PROPERTY proOnY_ITF : CtaSysIO.ITF_IO
GET
END_GET
END_PROPERTY

PROPERTY proIsRegulatet : BOOL
GET
END_GET
END_PROPERTY

PROPERTY proIsHandOnOrOff : BOOL
GET
END_GET
END_PROPERTY

PROPERTY proRunAfterTimeAktive : BOOL
GET
END_GET
END_PROPERTY

PROPERTY proLeadTimeAktive : BOOL
GET
END_GET
END_PROPERTY

PROPERTY proIsReady : BOOL
GET
END_GET
END_PROPERTY

PROPERTY proAuto : BOOL
GET
END_GET
SET
END_SET
END_PROPERTY

PROPERTY proHandOn : BOOL
SET
END_SET
GET
END_GET
END_PROPERTY

PROPERTY proIsError : BOOL
GET
END_GET
END_PROPERTY

PROPERTY proIsWarning : BOOL
GET
END_GET
END_PROPERTY

PROPERTY proEn : BOOL
GET
END_GET
SET
END_SET
END_PROPERTY

PROPERTY proHardWareHandModulAktive : BOOL
GET
END_GET
END_PROPERTY

PROPERTY proIsEnabled : BOOL
GET
END_GET
END_PROPERTY

PROPERTY proMotorIsOn : BOOL
GET
END_GET
END_PROPERTY

PROPERTY proHandOff : BOOL
SET
END_SET
GET
END_GET
END_PROPERTY

PROPERTY proRevisionSwitchOk : BOOL
GET
END_GET
END_PROPERTY

PROPERTY proHandOnY : REAL
SET
END_SET
GET
END_GET
END_PROPERTY

{attribute 'hide'} 
PROPERTY INTERNAL proEnSymbol : STRING
GET
END_GET
END_PROPERTY

PROPERTY proIsOn : BOOL
GET
END_GET
END_PROPERTY

PROPERTY proIsOnY : REAL
GET
END_GET
END_PROPERTY

PROPERTY proLeadTime : TIME
GET
END_GET
END_PROPERTY

PROPERTY proOn : BOOL
GET
END_GET
END_PROPERTY

PROPERTY proOnY : REAL
GET
END_GET
END_PROPERTY

PROPERTY proRunAfterTime : TIME
GET
END_GET
END_PROPERTY

{attribute 'hide'} 
PROPERTY INTERNAL proStateSymbol : STRING
GET
END_GET
END_PROPERTY

{attribute 'monitoring' := 'variable'}
PROPERTY proLockDown : BOOL
GET
END_GET
END_PROPERTY

{attribute 'monitoring' := 'variable'}
PROPERTY proAvailable : BOOL
GET
END_GET
END_PROPERTY

{attribute 'monitoring' := 'variable'}
PROPERTY proAcknowlege : BOOL
GET
END_GET
END_PROPERTY

PROPERTY proIconNr : UINT
SET
END_SET
GET
END_GET
END_PROPERTY

END_INTERFACE

// 30 Program Organization Units/fcGetBigerStringValue
FUNCTION fcGetBigerStringValue : INT
VAR_INPUT
    st1     :   STRING(255);
    st2     :   STRING(255);
END_VAR
VAR
    diFor: DINT;
    diMax: DINT;
END_VAR

IF LEN(st1) > LEN(st2) THEN
    diMax := LEN(st2); 
    fcGetBigerStringValue := 1;
ELSIF LEN(st1) < LEN(st2) THEN
    diMax := LEN(st1);
    fcGetBigerStringValue := 2;     
ELSE
    diMax := LEN(st1);    
END_IF;
FOR diFor := 0 TO  diMax DO
    IF st1[diFor] > st2[diFor] THEN
        fcGetBigerStringValue := 1;  
        EXIT; 
    ELSIF st1[diFor] < st2[diFor] THEN
        fcGetBigerStringValue := 2;  
        EXIT;
    END_IF;
END_FOR;

END_FUNCTION

// 30 Program Organization Units/fcCheckQuerryAndIconReturn
FUNCTION fcCheckQuerryAndIconReturn : BOOL
VAR_INPUT
	_ITF_IN			: 	ITF_ANTRIEB;
	_uiIconNr_IN	:	UINT;
END_VAR

IF __QUERYINTERFACE(_ITF_IN,_ITF_IN) THEN
	fcCheckQuerryAndIconReturn := TRUE;	
	_ITF_IN.proIconNr := _uiIconNr_IN;
ELSE
	fcCheckQuerryAndIconReturn :=  FALSE;
END_IF

END_FUNCTION

// 40 Visualizations/POPUP/POPUP_ANTRIEB
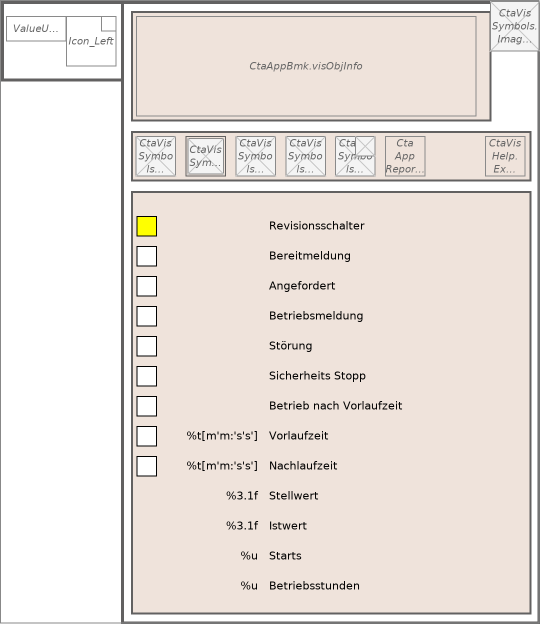
VISUALIZATION POPUP_ANTRIEB  // 540x624
VAR_INPUT
    ITF_ANTRIEBIN    	:   ITF_ANTRIEB;
	stExklParameter_IN	:	STRING[40];	
	uiPopUpGruppe 		: 	UINT;
END_VAR
    RoundedRectangle (1,1 160x80)
    RoundedRectangle (121,1 419x623)
    RoundedRectangle (131,11 360x110)
    Frame (136,16 340x100)
        shows CtaAppBmk.visObjInfo(ITF_BMK_IN := ITF_ANTRIEBIN)
    Image (490,1 50x50), image: CtaVisSymbols.ImagePool.close_solo_black
        OnMouseClick:  Dialog=POPUP_ANTRIEB, Result=None, NumpadKeypadSet=True
    Frame (6,16 110x50), input disabled if: TRUE, frame switch variable: ITF_ANTRIEBIN.proIconNr
        shows VIS_ANTRIEB_LEFT_ABOVE(ITF_ANTRIEB_IN := ITF_ANTRIEBIN, stExklParameter := stExklParameter_IN)
        shows VIS_ANTRIEB_LEFT_BELOW(ITF_ANTRIEB_IN := ITF_ANTRIEBIN, stExklParameter := stExklParameter_IN)
        shows VIS_ANTRIEB_RIGHT_ABOVE(ITF_ANTRIEB_IN := ITF_ANTRIEBIN, stExklParameter := stExklParameter_IN)
        shows VIS_ANTRIEB_RIGHT_BELOW(ITF_ANTRIEB_IN := ITF_ANTRIEBIN, stExklParameter := stExklParameter_IN)
    RoundedRectangle (131,191 400x423)
    Frame (132,206 398x400), frame switch variable: uiPopUpGruppe
        shows VIS_ANTRIEB_OVERVIEW(ITF_ANTRIEBIN := ITF_ANTRIEBIN)
        shows VIS_ANTRIEB_MANUAL(ITF_ANTRIEBIN := ITF_ANTRIEBIN)
        shows VIS_ANTRIEB_PARAMETER(ITF_ANTRIEBIN := ITF_ANTRIEBIN)
        shows VIS_ANTRIEB_IO(ITF_ANTRIEBIN := ITF_ANTRIEBIN)
        shows AT_BUS(ITF_ANTRIEBIN := ITF_ANTRIEBIN)
        shows VIS_ANTRIEB_REPORTS(ITF_ANTRIEBIN := ITF_ANTRIEBIN)
        pReferences[2]: ITF_Parameter=ITF_ANTRIEBIN.proParameter
    RoundedRectangle (131,131 400x50)
    Frame (131,136 399x40)
        shows VIS_ANTRIEB_LISTE(uiPopUpGruppe := uiPopUpGruppe, xHand := ITF_ANTRIEBIN.proIsHandOnOrOff, xHandOff := ITF_ANTRIEBIN.proHandOff, ITF_REPORTMANAGER_IN := ITF_ANTRIEBIN.proITF_REPORTMANAGER, xBusTestAktiv := ITF_ANTRIEBIN.proModbusTest, stExklParameter_IN := stExklParameter_IN)
    InvisibleInput (131,3 360x48)
END_VISUALIZATION

// 40 Visualizations/POPUP/VIS_ANTRIEB_LISTE
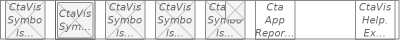
VISUALIZATION VIS_ANTRIEB_LISTE  // 400x40
VAR_IN_OUT
	uiPopUpGruppe 			:	UINT;
END_VAR
VAR_INPUT
    xHand           		: 	BOOL;
    xHandOff        		: 	BOOL;
    ITF_REPORTMANAGER_IN 	: 	CtaAppReport.ITF_REPORTMANAGER;
    xBusTestAktiv   		: 	BOOL;	
	stExklParameter_IN		:	STRING[40];
END_VAR
    Group (5,0 40x40)
        RoundedRectangle (0,0 40x40), colour toggle: uiPopUpGruppe = 0
            OnMouseDown: execute { uiPopUpGruppe := 0; }
        Image (0,0 40x40), image: CtaVisSymbols.ImagePool.eye
            OnMouseDown: execute { uiPopUpGruppe := 0; }
    Group (105,0 40x40)
        RoundedRectangle (0,0 40x40), colour toggle: uiPopUpGruppe = 2
            OnMouseDown: execute { uiPopUpGruppe := 2; }
        Image (0,0 40x40), image: CtaVisSymbols.ImagePool.gear
            OnMouseDown: execute { uiPopUpGruppe := 2; }
    Group (55,0 40x40)
        RoundedRectangle (0,0 40x40), colour toggle: uiPopUpGruppe = 1
            OnMouseDown: execute { uiPopUpGruppe := 1; }
        Image (2,2 36x36), image: CtaVisSymbols.ImagePool.front_hand_Black
            OnMouseDown: execute { uiPopUpGruppe := 1; }
        Image (2,2 36x36), invisible if: NOT xHand, image: CtaVisSymbols.ImagePool.front_hand_Yellow
            OnMouseDown: execute { uiPopUpGruppe := 1; }
        Image (2,2 36x36), invisible if: NOT xHandOff, image: CtaVisSymbols.ImagePool.front_hand_Yellow_Off
            OnMouseDown: execute { uiPopUpGruppe := 1; }
    Group (155,0 40x40)
        RoundedRectangle (0,0 40x40), colour toggle: uiPopUpGruppe = 3
            OnMouseDown: execute { uiPopUpGruppe := 3; }
        Image (0,0 40x40), image: CtaVisSymbols.ImagePool.dip-switch
            OnMouseDown: execute { uiPopUpGruppe := 3; }
    Group (205,0 40x40)
        RoundedRectangle (0,0 40x40), colour toggle: uiPopUpGruppe = 4
            OnMouseDown: execute { uiPopUpGruppe := 4; }
        Image (0,0 40x40), image: CtaVisSymbols.ImagePool.lan
            OnMouseDown: execute { uiPopUpGruppe := 4; }
        Image (20,0 20x20), invisible if: NOT xBusTestAktiv, image: CtaVisSymbols.ImagePool.front_hand_Yellow
            OnMouseDown: execute { uiPopUpGruppe := 4; }
    Group (255,0 40x40)
        RoundedRectangle (0,0 40x40), colour toggle: uiPopUpGruppe = 5
            OnMouseDown: execute { uiPopUpGruppe := 5; }
        Frame (0,0 40x40), input disabled if: TRUE
            shows CtaAppReport.VIS_ANZ_REPORTS_MODUL(ITF_REPORTMANAGER_IN := ITF_REPORTMANAGER_IN)
            OnMouseDown: execute { uiPopUpGruppe := 5; }
    Group (355,0 40x40)
        RoundedRectangle (0,0 40x40), invisible if: stExklParameter_IN = ' '
        Frame (0,0 40x40)
            shows CtaVisHelp.ExkParameterSymbol(stExklParameter := stExklParameter_IN)
END_VISUALIZATION

// 40 Visualizations/ICON/ANTRIEB_RIGHT/ANTRIEB_RIGHT_ABOVE/VIS_ANTRIEB_RigthAboveCheckQuerry
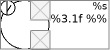
VISUALIZATION VIS_ANTRIEB_RigthAboveCheckQuerry  // 110x50
VAR_INPUT
    ITF_ANTRIEB_IN   :   ITF_ANTRIEB;	
END_VAR
VAR_INPUT
	stExklParameter		:	STRING[40];
END_VAR
    Frame (0,0 110x50)
        shows VIS_ANTRIEB_RigthAboveCheckIsEnabled(ITF_ANTRIEB_IN := ITF_ANTRIEB_IN, stExklParameter := stExklParameter)
END_VISUALIZATION

// 40 Visualizations/ICON/ANTRIEB_RIGHT/ANTRIEB_RIGHT_ABOVE/VIS_ANTRIEB_RIGHT_ABOVE
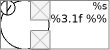
VISUALIZATION VIS_ANTRIEB_RIGHT_ABOVE  // 110x50
VAR_INPUT
    ITF_ANTRIEB_IN   :   ITF_ANTRIEB;	
END_VAR
VAR_INPUT CONSTANT
	stExklParameter		:	STRING[40] := ' ';
END_VAR
VAR CONSTANT
	uiIconNr		: UINT := 2;
END_VAR
    Frame (0,0 110x50), invisible if: NOT fcCheckQuerryAndIconReturn(_ITF_IN := ITF_ANTRIEB_IN, _uiIconNr_IN := uiIconNr)
        shows VIS_ANTRIEB_RigthAboveCheckQuerry(ITF_ANTRIEB_IN := ITF_ANTRIEB_IN, stExklParameter := stExklParameter)
END_VISUALIZATION

// 40 Visualizations/ICON/ANTRIEB_RIGHT/ANTRIEB_RIGHT_ABOVE/VIS_ANTRIEB_RigthAboveCheckIsEnabled
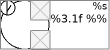
VISUALIZATION VIS_ANTRIEB_RigthAboveCheckIsEnabled  // 110x50
VAR_INPUT
    ITF_ANTRIEB_IN   :   ITF_ANTRIEB;	
END_VAR
VAR_INPUT
	stExklParameter		:	STRING[40];
END_VAR
    Frame (0,0 50x50), invisible if: NOT ITF_ANTRIEB_IN.proIsEnabled
        shows Icon_Right(ITF_ANTRIEB_IN := ITF_ANTRIEB_IN)
        shows Value_Right()
    Frame (50,0 60x25), invisible if: NOT ITF_ANTRIEB_IN.proIsEnabled
        shows ValueUpDwn(ITF_ANTRIEB_IN := ITF_ANTRIEB_IN, uiTextAusrichtung := 4)
    Frame (0,0 15x15), invisible if: NOT ITF_ANTRIEB_IN.proIsEnabled
        shows CommandOn(ITF_ANTRIEB_IN := ITF_ANTRIEB_IN)
    Rectangle (0,0 110x50)
        OnMouseClick:  Dialog=POPUP_ANTRIEB, Parameters={uiPopUpGruppe: 0, stExklParameter_IN: stExklParameter, ITF_ANTRIEBIN: ITF_ANTRIEB_IN}, OpenCentered=True
END_VISUALIZATION

// 40 Visualizations/ICON/ANTRIEB_BASE/CommandOn
VISUALIZATION CommandOn  // 15x15
VAR_INPUT
    ITF_ANTRIEB_IN   :   ITF_ANTRIEB;	
END_VAR
    Ellipse (0,0 15x15), colour toggle: ITF_ANTRIEB_IN.proOn
    Line (7,15) (7,10)
    Line (7,5) (7,0)
    Line (7,11) (11,5), invisible if: ITF_ANTRIEB_IN.proOn
    Line (7,15) (7,0), invisible if: NOT ITF_ANTRIEB_IN.proOn
END_VISUALIZATION

// 40 Visualizations/ICON/ANTRIEB_BASE/ICON/Icon_Left
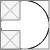
VISUALIZATION Icon_Left  // 50x50
VAR_INPUT
    ITF_ANTRIEB_IN   :   ITF_ANTRIEB;	
END_VAR
    Ellipse (0,0 49x49), colour toggle: ITF_ANTRIEB_IN.proMotorIsOn, invisible if: ITF_ANTRIEB_IN.proIsError
    Ellipse (0,0 49x49), colour toggle: ITF_ANTRIEB_IN.proIsError
    Image (0,0 20x20), invisible if: NOT ITF_ANTRIEB_IN.proIsWarning, image: CtaVisSymbols.ImagePool.CtaWarning
    Image (0,30 20x20), invisible if: NOT ITF_ANTRIEB_IN.proIsHandOnOrOff, image: CtaVisSymbols.ImagePool.front_hand_Yellow
    Image (0,30 20x20), invisible if: NOT ITF_ANTRIEB_IN.proHandOff, image: CtaVisSymbols.ImagePool.front_hand_Yellow_Off
END_VISUALIZATION

// 40 Visualizations/POPUP/PARAMETER/VIS_ANTRIEB_PARAMETER
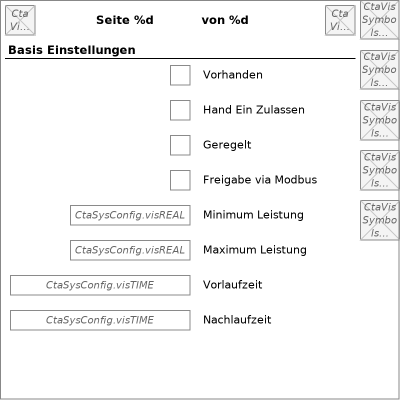
VISUALIZATION VIS_ANTRIEB_PARAMETER  // 400x400
VAR_INPUT
    ITF_ANTRIEBIN    :   ITF_ANTRIEB;	
END_VAR
VAR
    uiParameterGruppe : UINT;
END_VAR
    Frame (360,0 40x300)
        shows VIS_ANTRIEB_PARAMETER_LISTE(uiParameterGruppe := uiParameterGruppe)
    Frame (0,0 360x400), frame switch variable: uiParameterGruppe
        shows VIS_ANTRIEB_PARAMETER_BASE(ITF_ANTRIEBIN := ITF_ANTRIEBIN)
        shows VIS_ANTRIEB_PARAMETER_FUSES(ITF_ANTRIEBIN := ITF_ANTRIEBIN)
        shows VIS_ANTRIEB_PARAMETER_IO(ITF_ANTRIEBIN := ITF_ANTRIEBIN)
        shows VIS_ANTRIEB_PARAMETER_DATA(ITF_ANTRIEBIN := ITF_ANTRIEBIN)
        shows VIS_ANTRIEB_PARAMETER_TRENDLOG(ITF_ANTRIEBIN := ITF_ANTRIEBIN)
        pReferences[0]: ITF_Parameter=ITF_Parameter
        pReferences[1]: ITF_Parameter=ITF_Parameter
        pReferences[2]: ITF_Parameter=ITF_Parameter
        pReferences[3]: ITF_Parameter=ITF_Parameter
        pReferences[4]: ITF_Parameter=ITF_Parameter
END_VISUALIZATION

// 40 Visualizations/POPUP/PARAMETER/VIS_ANTRIEB_PARAMETER_LISTE
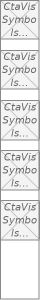
VISUALIZATION VIS_ANTRIEB_PARAMETER_LISTE  // 40x300
VAR_IN_OUT
	uiParameterGruppe : UINT;
END_VAR
    RoundedRectangle (0,150 39x39), colour toggle: uiParameterGruppe = 3
        OnMouseDown: execute { uiParameterGruppe := 3; }
    RoundedRectangle (0,100 39x39), colour toggle: uiParameterGruppe = 2
        OnMouseDown: execute { uiParameterGruppe := 2; }
    RoundedRectangle (0,50 39x39), colour toggle: uiParameterGruppe = 1
        OnMouseDown: execute { uiParameterGruppe := 1; }
    RoundedRectangle (0,0 39x39), colour toggle: uiParameterGruppe = 0
        OnMouseDown: execute { uiParameterGruppe := 0; }
    RoundedRectangle (0,200 39x39), colour toggle: uiParameterGruppe = 4
        OnMouseDown: execute { uiParameterGruppe := 4; }
    Image (0,0 39x39), image: CtaVisSymbols.ImagePool.engine
        OnMouseDown: execute { uiParameterGruppe := 0; }
    Image (0,50 39x39), image: CtaVisSymbols.ImagePool.electric_bolt_24dp_000000_FILL0_wght400_GRAD0_opsz24
        OnMouseDown: execute { uiParameterGruppe := 1; }
    Image (0,100 40x40), image: CtaVisSymbols.ImagePool.dip-switch
        OnMouseDown: execute { uiParameterGruppe := 2; }
    Image (0,150 40x40), image: CtaVisSymbols.ImagePool.database_black
        OnMouseDown: execute { uiParameterGruppe := 3; }
    Image (0,200 40x40), image: CtaVisSymbols.ImagePool.sine-wave
        OnMouseDown: execute { uiParameterGruppe := 4; }
END_VISUALIZATION

// 40 Visualizations/POPUP/MANUAL/VIS_ANTRIEB_MANUAL
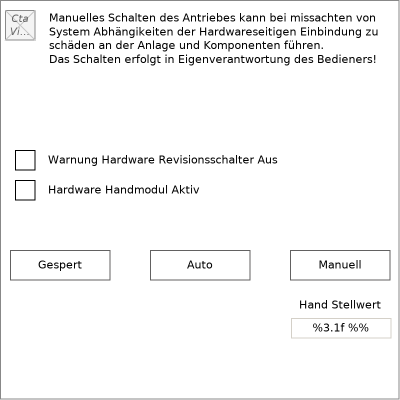
VISUALIZATION VIS_ANTRIEB_MANUAL  // 400x400
VAR_INPUT
    ITF_ANTRIEBIN    :   ITF_ANTRIEB;	
END_VAR
    Label (46,10 350x100), "Manuelles Schalten des Antriebes kann bei missachten von System Abhängikeiten der Hardwareseitigen Einbindung zu schäden an der Anlage und Komponenten führen. Das Schalten erfolgt in Eigenverantwortung des Bedieners!"
    Textfield (291,318 100x20), "%3.1f %%", text variable: ITF_ANTRIEBIN.proHandOnY, invisible if: NOT ITF_ANTRIEBIN.proIsRegulatet
        OnMouseClick: write the text variable via InputWithLimits, min 0, max 100, title 'Stellwert'
    Image (5,10 30x30), image: CtaVisSymbols.ImagePool.CtaWarning
    Label (290,295 100x20), "Hand Stellwert"
    Rectangle (15,180 20x20), colour toggle: ITF_ANTRIEBIN.proHardWareHandModulAktive, invisible if: NOT ITF_ANTRIEBIN.proHardWareHandModulAktive
    Label (45,180 200x20), "Hardware Handmodul Aktiv", invisible if: NOT ITF_ANTRIEBIN.proHardWareHandModulAktive
    Label (45,150 350x20), "Warnung Hardware Revisionsschalter Aus", invisible if: ITF_ANTRIEBIN.proRevisionSwitchOk
    Rectangle (15,150 20x20), colour toggle: NOT ITF_ANTRIEBIN.proRevisionSwitchOk, invisible if: ITF_ANTRIEBIN.proRevisionSwitchOk
    RoundedRectangle (10,250 100x30), "Gespert", colour toggle: ITF_ANTRIEBIN.proHandOff
        toggle ITF_ANTRIEBIN.proHandOff
    RoundedRectangle (150,250 100x30), "Auto", colour toggle: ITF_ANTRIEBIN.proAuto
        toggle ITF_ANTRIEBIN.proAuto
    RoundedRectangle (290,250 100x30), "Manuell", colour toggle: ITF_ANTRIEBIN.proHandOn
        toggle ITF_ANTRIEBIN.proHandOn
END_VISUALIZATION

// 40 Visualizations/POPUP/OVERVIEW/VIS_ANTRIEB_OVERVIEW
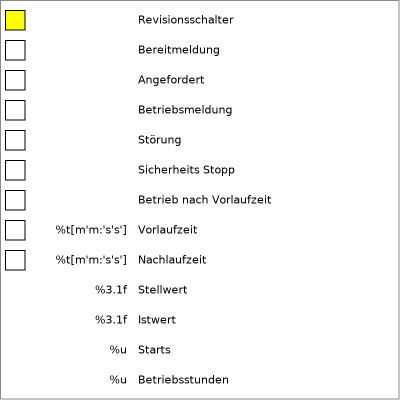
VISUALIZATION VIS_ANTRIEB_OVERVIEW  // 400x400
VAR_INPUT
    ITF_ANTRIEBIN    :   ITF_ANTRIEB;	
END_VAR
    Label (135,220 200x20), "Vorlaufzeit"
    Label (135,250 200x20), "Nachlaufzeit"
    Textfield (30,220 100x20), "%t[m'm:'s's']", text variable: ITF_ANTRIEBIN.proLeadTime
    Textfield (30,250 100x20), "%t[m'm:'s's']", text variable: ITF_ANTRIEBIN.proRunAfterTime
    Rectangle (5,220 20x20), colour toggle: ITF_ANTRIEBIN.proLeadTimeAktive
    Rectangle (5,250 20x20), colour toggle: ITF_ANTRIEBIN.proRunAfterTimeAktive
    Label (135,10 200x20), "Revisionsschalter"
    Label (135,40 200x20), "Bereitmeldung"
    Label (135,100 200x20), "Betriebsmeldung"
    Label (135,130 200x20), "Störung"
    Label (135,70 200x20), "Angefordert"
    Rectangle (5,10 20x20), colour toggle: ITF_ANTRIEBIN.proRevisionSwitchOk
    Rectangle (5,40 20x20), colour toggle: ITF_ANTRIEBIN.proIsReady
    Rectangle (5,70 20x20), colour toggle: ITF_ANTRIEBIN.proOn
    Rectangle (5,100 20x20), colour toggle: ITF_ANTRIEBIN.proMotorIsOn
    Rectangle (5,130 20x20), colour toggle: ITF_ANTRIEBIN.proIsError
    Label (135,160 200x20), "Sicherheits Stopp"
    Rectangle (5,160 20x20)
    Label (135,190 200x20), "Betrieb nach Vorlaufzeit"
    Rectangle (5,190 20x20), colour toggle: ITF_ANTRIEBIN.proIsOn
    Label (135,280 200x20), "Stellwert", invisible if: NOT ITF_ANTRIEBIN.proIsRegulatet
    Label (135,310 200x20), "Istwert", invisible if: NOT ITF_ANTRIEBIN.proIsRegulatet
    Textfield (30,280 100x20), "%3.1f", text variable: ITF_ANTRIEBIN.proOnY, invisible if: NOT ITF_ANTRIEBIN.proIsRegulatet
    Textfield (30,310 100x20), "%3.1f", text variable: ITF_ANTRIEBIN.proIsOnY, invisible if: NOT ITF_ANTRIEBIN.proIsRegulatet
    Textfield (30,370 100x20), "%u", text variable: ITF_ANTRIEBIN.proCountedHours
    Textfield (30,340 100x20), "%u", text variable: ITF_ANTRIEBIN.proCountedStarts
    Label (135,340 200x20), "Starts"
    Label (135,370 200x20), "Betriebsstunden"
END_VISUALIZATION

// 40 Visualizations/POPUP/BUS/AT_BUS
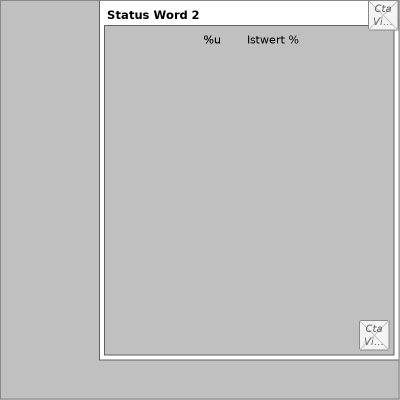
VISUALIZATION AT_BUS  // 400x400
VAR_INPUT
    ITF_ANTRIEBIN    :   ITF_ANTRIEB;	
END_VAR
    Frame (99,0 300x360)
        shows AT_BUS_CS(ITF_ANTRIEBIn := ITF_ANTRIEBIN, ayControllWord := ITF_ANTRIEBIN.proModbusControllWord, ayStateWord := ITF_ANTRIEBIN.proModbusStateWord)
END_VISUALIZATION

// 40 Visualizations/POPUP/BUS/AT_BUS_SW0_Detail
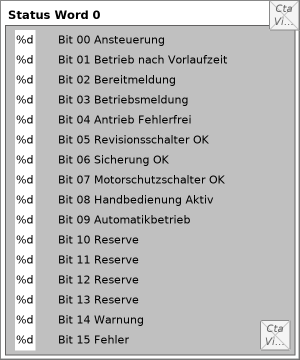
VISUALIZATION AT_BUS_SW0_Detail  // 300x360
VAR_IN_OUT
    wDetail     :   WORD;
END_VAR
VAR_INPUT	
    ITF_ANTRIEBIN    :   ITF_ANTRIEB;
END_VAR
VAR_IN_OUT
    xShow       :   BOOL;
END_VAR
    RoundedRectangle (0,0 300x360)
    RoundedRectangle (5,25 290x330)
    Textfield (15,30 20x20), "%d", text variable: TO_WORD(wDetail.0), input disabled if: NOT ITF_ANTRIEBIn.proModbusTest
        OnMouseClick: execute { wDetail.0 := NOT wDetail.0; }
    Label (55,30 220x20), "Bit 00 Ansteuerung"
    Textfield (15,50 20x20), "%d", text variable: TO_WORD(wDetail.1), input disabled if: NOT ITF_ANTRIEBIn.proModbusTest
        OnMouseClick: execute { wDetail.1 := NOT wDetail.1; }
    Label (55,50 220x20), "Bit 01 Betrieb nach Vorlaufzeit"
    Textfield (15,70 20x20), "%d", text variable: TO_WORD(wDetail.2), input disabled if: NOT ITF_ANTRIEBIn.proModbusTest
        OnMouseClick: execute { wDetail.2 := NOT wDetail.2; }
    Label (55,70 220x20), "Bit 02 Bereitmeldung"
    Textfield (15,90 20x20), "%d", text variable: TO_WORD(wDetail.3), input disabled if: NOT ITF_ANTRIEBIn.proModbusTest
        OnMouseClick: execute { wDetail.3 := NOT wDetail.3; }
    Label (55,90 220x20), "Bit 03 Betriebsmeldung"
    Textfield (15,110 20x20), "%d", text variable: TO_WORD(wDetail.4), input disabled if: NOT ITF_ANTRIEBIn.proModbusTest
        OnMouseClick: execute { wDetail.4 := NOT wDetail.4; }
    Label (55,110 220x20), "Bit 04 Antrieb Fehlerfrei"
    Textfield (15,130 20x20), "%d", text variable: TO_WORD(wDetail.5), input disabled if: NOT ITF_ANTRIEBIn.proModbusTest
        OnMouseClick: execute { wDetail.5 := NOT wDetail.5; }
    Label (55,130 220x20), "Bit 05 Revisionsschalter OK"
    Textfield (15,150 20x20), "%d", text variable: TO_WORD(wDetail.6), input disabled if: NOT ITF_ANTRIEBIn.proModbusTest
        OnMouseClick: execute { wDetail.6 := NOT wDetail.6; }
    Label (55,150 220x20), "Bit 06 Sicherung OK"
    Textfield (15,170 20x20), "%d", text variable: TO_WORD(wDetail.7), input disabled if: NOT ITF_ANTRIEBIn.proModbusTest
        OnMouseClick: execute { wDetail.7 := NOT wDetail.7; }
    Label (55,170 220x20), "Bit 07 Motorschutzschalter OK"
    Textfield (15,190 20x20), "%d", text variable: TO_WORD(wDetail.8), input disabled if: NOT ITF_ANTRIEBIn.proModbusTest
        OnMouseClick: execute { wDetail.8 := NOT wDetail.8; }
    Label (55,190 220x20), "Bit 08 Handbedienung Aktiv"
    Textfield (15,210 20x20), "%d", text variable: TO_WORD(wDetail.9), input disabled if: NOT ITF_ANTRIEBIn.proModbusTest
        OnMouseClick: execute { wDetail.9 := NOT wDetail.9; }
    Label (55,210 220x20), "Bit 09 Automatikbetrieb"
    Textfield (15,230 20x20), "%d", text variable: TO_WORD(wDetail.10), input disabled if: NOT ITF_ANTRIEBIn.proModbusTest
        OnMouseClick: execute { wDetail.10 := NOT wDetail.10; }
    Label (55,230 220x20), "Bit 10 Reserve"
    Textfield (15,250 20x20), "%d", text variable: TO_WORD(wDetail.11), input disabled if: NOT ITF_ANTRIEBIn.proModbusTest
        OnMouseClick: execute { wDetail.11 := NOT wDetail.11; }
    Label (55,250 220x20), "Bit 11 Reserve"
    Textfield (15,270 20x20), "%d", text variable: TO_WORD(wDetail.12), input disabled if: NOT ITF_ANTRIEBIn.proModbusTest
        OnMouseClick: execute { wDetail.12 := NOT wDetail.12; }
    Label (55,270 220x20), "Bit 12 Reserve"
    Textfield (15,290 20x20), "%d", text variable: TO_WORD(wDetail.13), input disabled if: NOT ITF_ANTRIEBIn.proModbusTest
        OnMouseClick: execute { wDetail.13 := NOT wDetail.13; }
    Label (55,290 220x20), "Bit 13 Reserve"
    Textfield (15,310 20x20), "%d", text variable: TO_WORD(wDetail.14), input disabled if: NOT ITF_ANTRIEBIn.proModbusTest
        OnMouseClick: execute { wDetail.14 := NOT wDetail.14; }
    Label (55,310 220x20), "Bit 14 Warnung"
    Textfield (15,330 20x20), "%d", text variable: TO_WORD(wDetail.15), input disabled if: NOT ITF_ANTRIEBIn.proModbusTest
        OnMouseClick: execute { wDetail.15 := NOT wDetail.15; }
    Label (55,330 220x20), "Bit 15 Fehler"
    Image (269,0 30x30), image: CtaVisSymbols.ImagePool.close_solo_black
        OnMouseClick: execute { xShow := FALSE; ITF_ANTRIEBIN.proModbusTest := FALSE; }
    Label (5,0 150x30), "Status Word 0"
    Image (260,320 30x30), invisible if: ITF_ANTRIEBIN.proModbusTest, image: CtaVisSymbols.ImagePool.front_hand_Black
        OnMouseClick: execute { ITF_ANTRIEBIN.proModbusTest := TRUE; }
    Image (260,320 30x30), invisible if: NOT ITF_ANTRIEBIN.proModbusTest, image: CtaVisSymbols.ImagePool.front_hand_Yellow
        OnMouseClick: execute { ITF_ANTRIEBIN.proModbusTest := False; }
END_VISUALIZATION

// 40 Visualizations/POPUP/BUS/AT_BUS_CW0_Detail
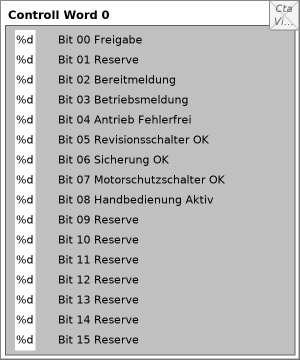
VISUALIZATION AT_BUS_CW0_Detail  // 300x360
VAR_IN_OUT
    wDetail :   WORD;
END_VAR
VAR_IN_OUT
    xShow   :   BOOL;
END_VAR
    RoundedRectangle (0,0 300x360)
    RoundedRectangle (5,25 290x330)
    Textfield (15,30 20x20), "%d", text variable: TO_WORD(wDetail.0), input disabled if: TRUE
    Label (55,30 180x20), "Bit 00 Freigabe"
    Textfield (15,50 20x20), "%d", text variable: TO_WORD(wDetail.1), input disabled if: TRUE
    Label (55,50 180x20), "Bit 01 Reserve"
    Textfield (15,70 20x20), "%d", text variable: TO_WORD(wDetail.2), input disabled if: TRUE
    Label (55,70 180x20), "Bit 02 Bereitmeldung"
    Textfield (15,90 20x20), "%d", text variable: TO_WORD(wDetail.3), input disabled if: TRUE
    Label (55,90 180x20), "Bit 03 Betriebsmeldung"
    Textfield (15,110 20x20), "%d", text variable: TO_WORD(wDetail.4), input disabled if: TRUE
    Label (55,110 180x20), "Bit 04 Antrieb Fehlerfrei"
    Textfield (15,130 20x20), "%d", text variable: TO_WORD(wDetail.5), input disabled if: TRUE
    Label (55,130 180x20), "Bit 05 Revisionsschalter OK"
    Textfield (15,150 20x20), "%d", text variable: TO_WORD(wDetail.6), input disabled if: TRUE
    Label (55,150 180x20), "Bit 06 Sicherung OK"
    Textfield (15,170 20x20), "%d", text variable: TO_WORD(wDetail.7), input disabled if: TRUE
    Label (55,170 180x20), "Bit 07 Motorschutzschalter OK"
    Textfield (15,190 20x20), "%d", text variable: TO_WORD(wDetail.8), input disabled if: TRUE
    Label (55,190 180x20), "Bit 08 Handbedienung Aktiv"
    Textfield (15,210 20x20), "%d", text variable: TO_WORD(wDetail.9), input disabled if: TRUE
    Label (55,210 180x20), "Bit 09 Reserve"
    Textfield (15,230 20x20), "%d", text variable: TO_WORD(wDetail.10), input disabled if: TRUE
    Label (55,230 180x20), "Bit 10 Reserve"
    Textfield (15,250 20x20), "%d", text variable: TO_WORD(wDetail.11), input disabled if: TRUE
    Label (55,250 180x20), "Bit 11 Reserve"
    Textfield (15,270 20x20), "%d", text variable: TO_WORD(wDetail.12), input disabled if: TRUE
    Label (55,270 180x20), "Bit 12 Reserve"
    Textfield (15,290 20x20), "%d", text variable: TO_WORD(wDetail.13), input disabled if: TRUE
    Label (55,290 180x20), "Bit 13 Reserve"
    Textfield (15,310 20x20), "%d", text variable: TO_WORD(wDetail.14), input disabled if: TRUE
    Label (55,310 180x20), "Bit 14 Reserve"
    Textfield (15,330 20x20), "%d", text variable: TO_WORD(wDetail.15), input disabled if: TRUE
    Label (55,330 180x20), "Bit 15 Reserve"
    Image (269,0 30x30), image: CtaVisSymbols.ImagePool.close_solo_black
        OnMouseClick: execute { xShow := FALSE; }
    Label (5,0 150x30), "Controll Word 0"
END_VISUALIZATION

// 40 Visualizations/POPUP/BUS/AT_BUS_CS
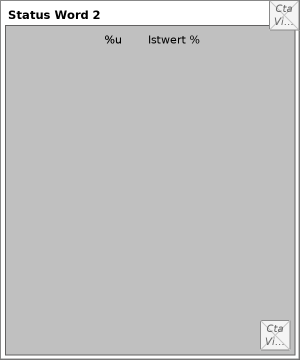
VISUALIZATION AT_BUS_CS  // 300x360
VAR_INPUT
    ITF_ANTRIEBIn        :   ITF_ANTRIEB;
    ayControllWord  :   REFERENCE TO ARRAY[0..3] OF WORD;
    ayStateWord     :   REFERENCE TO ARRAY[0..3] OF WORD;
END_VAR
VAR
    xShowCw :   BOOL;
    xShowSw :   BOOL;
    xShowSw1:   BOOL;
    xShowSw2:   BOOL;
END_VAR
    Textfield (0,10 130x20), "%b", text variable: ayControllWord[0]
    Label (140,10 120x20), "Controll Word 0"
    Label (140,50 120x20), "Controll Word 1"
    Textfield (0,50 130x20), "%d", text variable: ayControllWord[1]
    Label (140,90 120x20), "Controll Word 2", invisible if: TRUE
    Textfield (0,90 130x20), "%d", text variable: ayControllWord[2], invisible if: TRUE
    Label (140,130 120x20), "Controll Word 3", invisible if: TRUE
    Textfield (0,130 130x20), "%d", text variable: ayControllWord[2], invisible if: TRUE
    Image (265,5 30x30), image: CtaVisSymbols.ImagePool.information-variant
        OnMouseClick: execute {
            xShowCw := TRUE;
            xShowSw := FALSE;
            xShowSw1:= FALSE;
            xShowSw2:= FALSE;
        }
    Label (140,290 120x20), "State Word 3", invisible if: TRUE
    Textfield (0,170 130x20), "%b", text variable: ayStateWord[0]
        OnMouseDown: write the text variable via Default
    Label (140,170 120x20), "State Word 0"
    Label (140,210 120x20), "State Word 1"
    Textfield (0,210 130x20), "%d", text variable: ayStateWord[1]
    Label (140,250 120x20), "State Word 2"
    Textfield (0,250 130x20), "%d", text variable: ayStateWord[2]
    Textfield (0,290 130x20), "%d", text variable: ayStateWord[2], invisible if: TRUE
    Image (265,165 30x30), image: CtaVisSymbols.ImagePool.information-variant
        OnMouseClick: execute {
            xShowCw := FALSE;
            xShowSw := TRUE;
            xShowSw1:= FALSE;
            xShowSw2:= FALSE;
        }
    Image (265,205 30x30), image: CtaVisSymbols.ImagePool.information-variant
        OnMouseClick: execute {
            xShowCw := FALSE;
            xShowSw := FALSE;
            xShowSw1:= TRUE;
            xShowSw2:= FALSE;
        }
    Image (265,245 30x30), image: CtaVisSymbols.ImagePool.information-variant
        OnMouseClick: execute {
            xShowCw := FALSE;
            xShowSw := FALSE;
            xShowSw1:= FALSE;
            xShowSw2:= TRUE;
        }
    Frame (0,0 300x360), invisible if: NOT xShowCw
        shows AT_BUS_CW0_Detail(wDetail := ayControllWord[0], xShow := xShowCw)
    Frame (0,0 300x360), invisible if: NOT xShowSw
        shows AT_BUS_SW0_Detail(wDetail := ayStateWord[0], ITF_ANTRIEBIn := ITF_ANTRIEBIn, xShow := xShowSw)
        pReferences[0]: ITF_ATIn=ITF_ATIn
    Frame (0,0 300x360), invisible if: NOT xShowSw1
        shows AT_BUS_SW1_Detail(wDetail := ayStateWord[1], ITF_ANTRIEBIn := ITF_ANTRIEBIn, xShow := xShowSw1)
    Frame (0,0 300x360), invisible if: NOT xShowSw2
        shows AT_BUS_SW2_Detail(wDetail := ayStateWord[2], ITF_ANTRIEBIn := ITF_ANTRIEBIn, xShow := xShowSw2)
END_VISUALIZATION

// 40 Visualizations/POPUP/BUS/AT_BUS_SW1_Detail
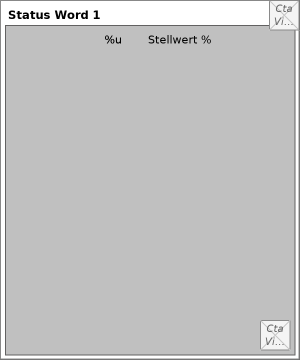
VISUALIZATION AT_BUS_SW1_Detail  // 300x360
VAR_IN_OUT
    wDetail     :   WORD;
END_VAR
VAR_INPUT	
    ITF_ANTRIEBIN    :   ITF_ANTRIEB;
END_VAR
VAR_IN_OUT
    xShow       :   BOOL;
END_VAR
    RoundedRectangle (0,0 300x360)
    RoundedRectangle (5,25 290x330)
    Image (269,0 30x30), image: CtaVisSymbols.ImagePool.close_solo_black
        OnMouseClick: execute { xShow := FALSE; ITF_ANTRIEBIN.proModbusTest := FALSE; }
    Label (5,0 150x30), "Status Word 1"
    Label (145,30 120x20), "Stellwert %"
    Textfield (15,30 110x20), "%u", text variable: wDetail, input disabled if: NOT ITF_ANTRIEBIn.proModbusTest
        OnMouseClick: write the text variable via InputWithLimits, min 0, max 100
    Textfield (15,30 110x20), "%u", text variable: wDetail, invisible if: ITF_ANTRIEBIN.proModbusTest
    Image (260,320 30x30), invisible if: ITF_ANTRIEBIN.proModbusTest, image: CtaVisSymbols.ImagePool.front_hand_Black
        OnMouseClick: execute { ITF_ANTRIEBIN.proModbusTest := TRUE; }
    Image (260,320 30x30), invisible if: NOT ITF_ANTRIEBIn.proModbusTest, image: CtaVisSymbols.ImagePool.front_hand_Yellow
        OnMouseClick: execute { ITF_ANTRIEBIN.proModbusTest := False; }
END_VISUALIZATION

// 40 Visualizations/POPUP/BUS/AT_BUS_SW2_Detail
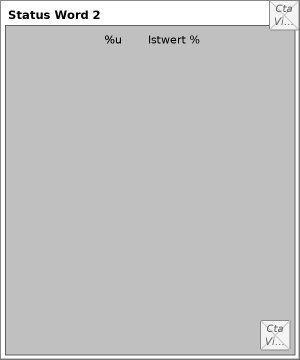
VISUALIZATION AT_BUS_SW2_Detail  // 300x360
VAR_IN_OUT
    wDetail             :   WORD;
END_VAR
VAR_INPUT	
    ITF_ANTRIEBIN       :   ITF_ANTRIEB;
END_VAR
VAR_IN_OUT
    xShow               :   BOOL;
END_VAR
    RoundedRectangle (0,0 300x360)
    RoundedRectangle (5,25 290x330)
    Image (269,0 30x30), image: CtaVisSymbols.ImagePool.close_solo_black
        OnMouseClick: execute { xShow := FALSE; ITF_ANTRIEBIN.proModbusTest := FALSE; }
    Label (5,0 150x30), "Status Word 2"
    Label (145,30 120x20), "Istwert %"
    Textfield (15,30 110x20), "%u", text variable: wDetail, input disabled if: NOT ITF_ANTRIEBIn.proModbusTest
        OnMouseClick: write the text variable via InputWithLimits, min 0, max 100
    Textfield (15,30 110x20), "%u", text variable: wDetail, invisible if: ITF_ANTRIEBIN.proModbusTest
    Image (260,320 30x30), invisible if: ITF_ANTRIEBIn.proModbusTest, image: CtaVisSymbols.ImagePool.front_hand_Black
        OnMouseClick: execute { ITF_ANTRIEBIN.proModbusTest := TRUE; }
    Image (260,320 30x30), invisible if: NOT ITF_ANTRIEBIN.proModbusTest, image: CtaVisSymbols.ImagePool.front_hand_Yellow
        OnMouseClick: execute { ITF_ANTRIEBIN.proModbusTest := False; }
END_VISUALIZATION

// 40 Visualizations/POPUP/REPORTS/VIS_ANTRIEB_REPORTS
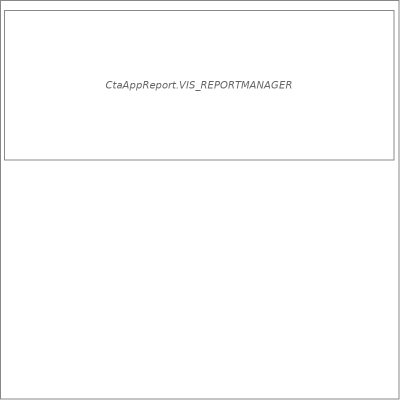
VISUALIZATION VIS_ANTRIEB_REPORTS  // 400x400
VAR_INPUT
    ITF_ANTRIEBIN    :   ITF_ANTRIEB;	
END_VAR
    Frame (4,10 390x150)
        shows CtaAppReport.VIS_REPORTMANAGER(ITF_REPORTMANAGER := ITF_ANTRIEBIN.proITF_REPORTMANAGER)
END_VISUALIZATION

// 40 Visualizations/POPUP/PARAMETER/AT_ParameterBase/VIS_ANTRIEB_PARAMETER_BASE0
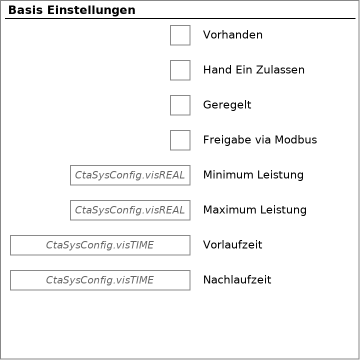
VISUALIZATION VIS_ANTRIEB_PARAMETER_BASE0  // 360x360
VAR_INPUT
    ITF_ANTRIEBIN    :   ITF_ANTRIEB;	
END_VAR
    Label (5,0 350x20), "Basis Einstellungen"
    Line (5,18) (355,18)
    Frame (170,25 20x20)
        shows CtaSysConfig.visBOOL(visfbBOOLIn := ITF_ANTRIEBIN.P_scBase_fbxEnable)
    Label (200,25 150x20), "Vorhanden"
    Frame (170,95 20x20)
        shows CtaSysConfig.visBOOL(visfbBOOLIn := ITF_ANTRIEBIN.P_scBase_fbxRegulatet)
    Label (200,95 150x20), "Geregelt"
    Frame (170,130 20x20)
        shows CtaSysConfig.visBOOL(visfbBOOLIn := ITF_ANTRIEBIN.P_scBase_fbxControllMb)
    Label (200,130 150x20), "Freigabe via Modbus"
    Frame (70,165 120x20)
        shows CtaSysConfig.visREAL(visfbREALIn := ITF_ANTRIEBIN.P_scBase_fbrYMin, stPhysikalischeEinheit := '%')
    Label (200,165 150x20), "Minimum Leistung"
    Frame (70,200 120x20)
        shows CtaSysConfig.visREAL(visfbREALIn := ITF_ANTRIEBIN.P_scBase_fbrYMax, stPhysikalischeEinheit := '%')
    Label (200,200 150x20), "Maximum Leistung"
    Frame (10,235 180x20)
        shows CtaSysConfig.visTIME(visfbTIMEIn := ITF_ANTRIEBIN.P_scBase_fbtLeadTime)
    Label (200,235 150x20), "Vorlaufzeit"
    Label (200,270 150x20), "Nachlaufzeit"
    Frame (10,270 180x20)
        shows CtaSysConfig.visTIME(visfbTIMEIn := ITF_ANTRIEBIN.P_scBase_fbtRunAfterTime)
    Frame (170,60 20x20)
        shows CtaSysConfig.visBOOL(visfbBOOLIn := ITF_ANTRIEBIN.P_scManual_fbxAlowManualOn)
    Label (200,60 150x20), "Hand Ein Zulassen"
END_VISUALIZATION

// 40 Visualizations/POPUP/PARAMETER/AT_ParameterBase/VIS_ANTRIEB_PARAMETER_BASE
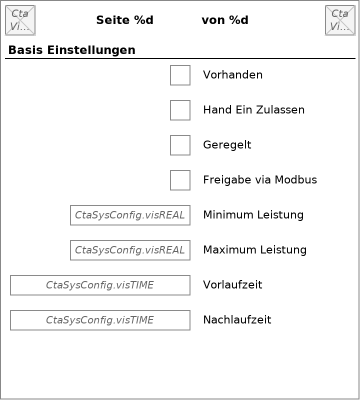
VISUALIZATION VIS_ANTRIEB_PARAMETER_BASE  // 360x400
VAR_INPUT
    ITF_ANTRIEBIN    :   ITF_ANTRIEB;	
END_VAR
VAR
    uiPage  :   UINT;
    uiMin   :   UINT    := 0;
    uiMax   :   UINT    := 0;
END_VAR
    Image (5,5 30x30), invisible if: uiPage = uiMin, image: CtaVisSymbols.ImagePool.arrow-left_square
        OnMouseClick: execute {
            uiPage := uiPage - 1;
            IF uiPage <= uiMin THEN
                uiPage := uiMin;
            END_IF;
        }
    Image (325,5 30x30), invisible if: uiPage = uiMax, image: CtaVisSymbols.ImagePool.arrow-right_square
        OnMouseClick: execute {
            uiPage := uiPage + 1;
            IF uiPage >= uiMax THEN
                uiPage := uiMax;
            END_IF;
        }
    Frame (0,40 360x360), frame switch variable: uiPage
        shows VIS_ANTRIEB_PARAMETER_BASE0(ITF_ANTRIEBIN := ITF_ANTRIEBIN)
        shows AT_ParameterIO1(ITF_Parameter := ITF_Parameter)
        pReferences[0]: ITF_Parameter=ITF_Parameter
    Textfield (175,5 100x30), "von %d", text variable: uiMax
    Textfield (75,5 100x30), "Seite %d", text variable: uiPage
END_VISUALIZATION

// 40 Visualizations/POPUP/PARAMETER/AT_Data/VIS_ANTRIEB_PARAMETER_DATA0
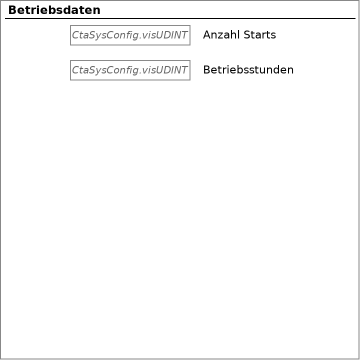
VISUALIZATION VIS_ANTRIEB_PARAMETER_DATA0  // 360x360
VAR_INPUT
    ITF_ANTRIEBIN    :   ITF_ANTRIEB;	
END_VAR
    Label (200,25 150x20), "Anzahl Starts"
    Label (200,60 150x20), "Betriebsstunden"
    Label (5,0 350x20), "Betriebsdaten"
    Frame (70,25 120x20)
        shows CtaSysConfig.visUDINT(visfbUDINTIn := ITF_ANTRIEBIN.P_scData_fbudiOperationStarts)
    Frame (70,60 120x20)
        shows CtaSysConfig.visUDINT(visfbUDINTIn := ITF_ANTRIEBIN.P_scData_fbudiOperatingHours)
    Line (5,18) (355,18)
END_VISUALIZATION

// 40 Visualizations/POPUP/PARAMETER/AT_Data/VIS_ANTRIEB_PARAMETER_DATA
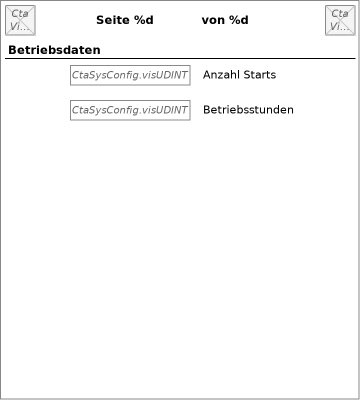
VISUALIZATION VIS_ANTRIEB_PARAMETER_DATA  // 360x400
VAR_INPUT
    ITF_ANTRIEBIN    :   ITF_ANTRIEB;	
END_VAR
VAR
    uiPage  :   UINT;
    uiMin   :   UINT    := 0;
    uiMax   :   UINT    := 0;
END_VAR
    Image (5,5 30x30), invisible if: uiPage = uiMin, image: CtaVisSymbols.ImagePool.arrow-left_square
        OnMouseClick: execute {
            uiPage := uiPage - 1;
            IF uiPage <= uiMin THEN
                uiPage := uiMin;
            END_IF;
        }
    Image (325,5 30x30), invisible if: uiPage = uiMax, image: CtaVisSymbols.ImagePool.arrow-right_square
        OnMouseClick: execute {
            uiPage := uiPage + 1;
            IF uiPage >= uiMax THEN
                uiPage := uiMax;
            END_IF;
        }
    Frame (0,40 360x360), frame switch variable: uiPage
        shows VIS_ANTRIEB_PARAMETER_DATA0(ITF_ANTRIEBIN := ITF_ANTRIEBIN)
        shows AT_ParameterIO1(ITF_Parameter := ITF_Parameter)
        pReferences[0]: ITF_Parameter=ITF_Parameter
    Textfield (75,5 100x30), "Seite %d", text variable: uiPage
    Textfield (175,5 100x30), "von %d", text variable: uiMax
END_VISUALIZATION

// 40 Visualizations/POPUP/PARAMETER/AT_Fuse/VIS_ANTRIEB_PARAMETER_FUSES0
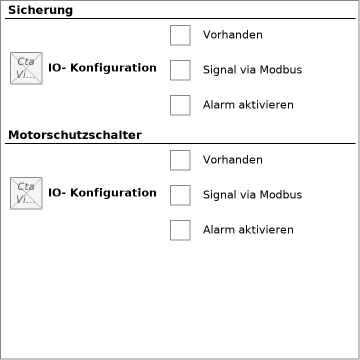
VISUALIZATION VIS_ANTRIEB_PARAMETER_FUSES0  // 360x360
VAR_INPUT
    ITF_ANTRIEBIN  		:	ITF_ANTRIEB;
	ITF_Fuse_IN			:	CtaSysIO.ITF_IO;
	ITF_MotorFuse_IN	:	CtaSysIO.ITF_IO;
END_VAR
    Frame (170,25 20x20)
        shows CtaSysConfig.visBOOL(visfbBOOLIn := ITF_ANTRIEBIN.P_scFuse_fbxEnable)
    Label (200,25 150x20), "Vorhanden"
    Frame (170,60 20x20)
        shows CtaSysConfig.visBOOL(visfbBOOLIn := ITF_ANTRIEBIN.P_scFuse_fbxInputMb)
    Label (200,60 150x20), "Signal via Modbus"
    Frame (170,95 20x20)
        shows CtaSysConfig.visBOOL(visfbBOOLIn := ITF_ANTRIEBIN.P_scFuse_fbxDoesAlarm)
    Label (200,95 150x20), "Alarm aktivieren"
    Label (5,0 350x20), "Sicherung"
    Label (5,125 350x20), "Motorschutzschalter"
    Frame (170,150 20x20)
        shows CtaSysConfig.visBOOL(visfbBOOLIn := ITF_ANTRIEBIN.P_scMotorFuse_fbxEnable)
    Label (200,150 150x20), "Vorhanden"
    Frame (170,185 20x20)
        shows CtaSysConfig.visBOOL(visfbBOOLIn := ITF_ANTRIEBIN.P_scMotorFuse_fbxInputMb)
    Label (200,185 150x20), "Signal via Modbus"
    Frame (170,220 20x20)
        shows CtaSysConfig.visBOOL(visfbBOOLIn := ITF_ANTRIEBIN.P_scMotorFuse_fbxDoesAlarm)
    Label (200,220 150x20), "Alarm aktivieren"
    Line (5,18) (355,18)
    Line (5,143) (355,143)
    Image (10,52 32x32), invisible if: ITF_Fuse_IN = 0, image: CtaVisSymbols.ImagePool.build
        OnMouseDown:  Dialog=VIS_ANTRIEB_POPUP_IO_ITF, Parameters={ITF_IO_IN: ITF_Fuse_IN}, OpenModal=True, OpenCentered=True
    Image (10,177 32x32), invisible if: ITF_MotorFuse_IN = 0, image: CtaVisSymbols.ImagePool.build
        OnMouseDown:  Dialog=VIS_ANTRIEB_POPUP_IO_ITF, Parameters={ITF_IO_IN: ITF_MotorFuse_IN}, OpenModal=True, OpenCentered=True
    Label (45,58 120x20), "IO- Konfiguration", invisible if: ITF_Fuse_IN = 0
    Label (45,183 120x20), "IO- Konfiguration", invisible if: ITF_MotorFuse_IN = 0
END_VISUALIZATION

// 40 Visualizations/POPUP/PARAMETER/AT_Fuse/VIS_ANTRIEB_PARAMETER_FUSES
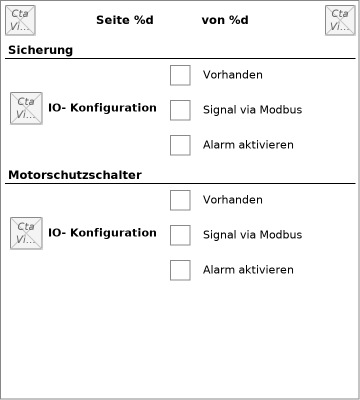
VISUALIZATION VIS_ANTRIEB_PARAMETER_FUSES  // 360x400
VAR_INPUT
    ITF_ANTRIEBIN    :   ITF_ANTRIEB;	
END_VAR
VAR
    uiPage  :   UINT;
    uiMin   :   UINT    := 0;
    uiMax   :   UINT    := 0;
END_VAR
    Image (5,5 30x30), invisible if: uiPage = uiMin, image: CtaVisSymbols.ImagePool.arrow-left_square
        OnMouseClick: execute {
            uiPage := uiPage - 1;
            IF uiPage <= uiMin THEN
                uiPage := uiMin;
            END_IF;
        }
    Image (325,5 30x30), invisible if: uiPage = uiMax, image: CtaVisSymbols.ImagePool.arrow-right_square
        OnMouseClick: execute {
            uiPage := uiPage + 1;
            IF uiPage >= uiMax THEN
                uiPage := uiMax;
            END_IF;
        }
    Frame (0,40 360x360), frame switch variable: uiPage
        shows VIS_ANTRIEB_PARAMETER_FUSES0(ITF_ANTRIEBIN := ITF_ANTRIEBIN, ITF_Fuse_IN := ITF_ANTRIEBIN.proFuse_ITF, ITF_MotorFuse_IN := ITF_ANTRIEBIN.proMotorFuse_ITF)
        shows AT_ParameterIO1(ITF_Parameter := ITF_Parameter)
        pReferences[0]: ITF_Parameter=ITF_Parameter
    Textfield (75,5 100x30), "Seite %d", text variable: uiPage
    Textfield (175,5 100x30), "von %d", text variable: uiMax
END_VISUALIZATION

// 40 Visualizations/POPUP/PARAMETER/AT_IO/VIS_ANTRIEB_PARAMETER_IO0
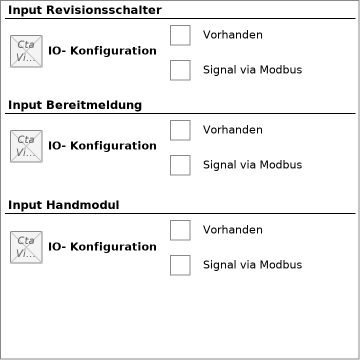
VISUALIZATION VIS_ANTRIEB_PARAMETER_IO0  // 360x360
VAR_INPUT
    ITF_ANTRIEBIN    	:   ITF_ANTRIEB;
	ITF_RevSwitch_IN	:	CtaSysIO.ITF_IO;
	ITF_Ready_IN		:	CtaSysIO.ITF_IO;
	ITF_HandModul_IN	:	CtaSysIO.ITF_IO;
END_VAR
    Frame (170,25 20x20)
        shows CtaSysConfig.visBOOL(visfbBOOLIn := ITF_ANTRIEBIN.P_scIO_RevisionSwitch_fbxEnable)
    Label (200,25 150x20), "Vorhanden"
    Frame (170,60 20x20)
        shows CtaSysConfig.visBOOL(visfbBOOLIn := ITF_ANTRIEBIN.P_scIO_RevisionSwitch_fbxInputMb)
    Label (200,60 150x20), "Signal via Modbus"
    Label (5,0 350x20), "Input Revisionsschalter"
    Label (5,95 350x20), "Input Bereitmeldung"
    Frame (170,120 20x20)
        shows CtaSysConfig.visBOOL(visfbBOOLIn := ITF_ANTRIEBIN.P_scIO_IsReady_fbxEnable)
    Label (200,120 150x20), "Vorhanden"
    Frame (170,155 20x20)
        shows CtaSysConfig.visBOOL(visfbBOOLIn := ITF_ANTRIEBIN.P_scIO_IsReady_fbxInputMb)
    Label (200,155 150x20), "Signal via Modbus"
    Label (5,195 350x20), "Input Handmodul"
    Frame (170,220 20x20)
        shows CtaSysConfig.visBOOL(visfbBOOLIn := ITF_ANTRIEBIN.P_scIO_IsHand_fbxEnable)
    Label (200,220 150x20), "Vorhanden"
    Frame (170,255 20x20)
        shows CtaSysConfig.visBOOL(visfbBOOLIn := ITF_ANTRIEBIN.P_scIO_IsHand_fbxInputMb)
    Label (200,255 150x20), "Signal via Modbus"
    Line (5,213) (355,213)
    Line (5,113) (355,113)
    Line (5,18) (355,18)
    Image (10,35 32x32), invisible if: ITF_RevSwitch_IN = 0, image: CtaVisSymbols.ImagePool.build
        OnMouseClick:  Dialog=VIS_ANTRIEB_POPUP_IO_ITF, Parameters={ITF_IO_IN: ITF_RevSwitch_IN}, OpenModal=True, OpenCentered=True
    Label (45,41 120x20), "IO- Konfiguration", invisible if: ITF_RevSwitch_IN = 0
    Image (10,130 32x32), invisible if: ITF_Ready_IN = 0, image: CtaVisSymbols.ImagePool.build
        OnMouseClick:  Dialog=VIS_ANTRIEB_POPUP_IO_ITF, Parameters={ITF_IO_IN: ITF_Ready_IN}, OpenModal=True, OpenCentered=True
    Label (45,136 120x20), "IO- Konfiguration", invisible if: ITF_Ready_IN = 0
    Image (10,231 32x32), invisible if: ITF_HandModul_IN = 0, image: CtaVisSymbols.ImagePool.build
        OnMouseClick:  Dialog=VIS_ANTRIEB_POPUP_IO_ITF, Parameters={ITF_IO_IN: ITF_HandModul_IN}, OpenModal=True, OpenCentered=True
    Label (45,237 120x20), "IO- Konfiguration", invisible if: ITF_HandModul_IN = 0
END_VISUALIZATION

// 40 Visualizations/POPUP/PARAMETER/AT_IO/VIS_ANTRIEB_PARAMETER_IO1
